PROGRAM MAIN
VAR
END_VAR

POU_Mdbus();

END_PROGRAM

(* stored: Version 1.1.0.1, ProductVersion 3.1.4024.12
   POU MAIN: Id {4a82918b-1a79-487e-bf49-41eb2f0c4ef8}, SpecialFunc None *)
